// TIA Portal project "PID_PROCCESS_CONTROL" (V16)

(* hardware
DEVICE "S7-1200 station_1"  S7-1200 Station
   slot 0: "Rack_0"  S7-1200 Rack  Rack  V1.0
   slot 1: "PLC_1"  CPU 1214C DC/DC/DC  6ES7 214-1AG40-0XB0  V4.4
   slot 2: "AI 4x13BIT/AQ 2x14BIT_1"  6ES7 234-4HE32-0XB0  V2.1
*)

// ===== PLC "PLC_1"  CPU 1214C DC/DC/DC =====

VAR_GLOBAL   // PLC tag table "Default tag table"
   "Tag_1" AT %MD2 : DWord;
   "Tag_2" AT %M500.0 : Bool;
   "Tag_3" AT %MD67 : Real;
   "Tag_4" AT %MD77 : DWord;
   "SP" AT %MD96 : Real;
   "Tag_5" AT %Q0.3 : Bool;
   "Tag_6" AT %MD70 : Real;
END_VAR

VAR_GLOBAL   // PLC tag table "INPUTS&OUTPUTS"
   "PRESSURE_SENSOR" AT %IW64 : Int;
   "FLOW_VALVE" AT %QW96 : Int;
   "SWITCH_1" AT %I0.1 : Bool;
   "SWITCH_2_SOLENOID" AT %I0.2 : Bool;
   "PUMP" AT %Q0.0 : Bool;
   "SOLENOID" AT %Q0.1 : Bool;
   "STORE_MEM" AT %MD20 : DWord;
   "FINAL_VAL" AT %MD30 : DWord;
END_VAR

ORGANIZATION_BLOCK "Main"   // OB1, LAD, ProgramCycle
TITLE = "Main Program Sweep (Cycle)"
{ S7_Optimized_Access := 'TRUE' }
VERSION : 0.1
   VAR_INPUT
      Initial_Call : Bool;   // Initial call of this OB
      Remanence : Bool;   // =True, if remanent data are available
   END_VAR
BEGIN

REGION Network 1
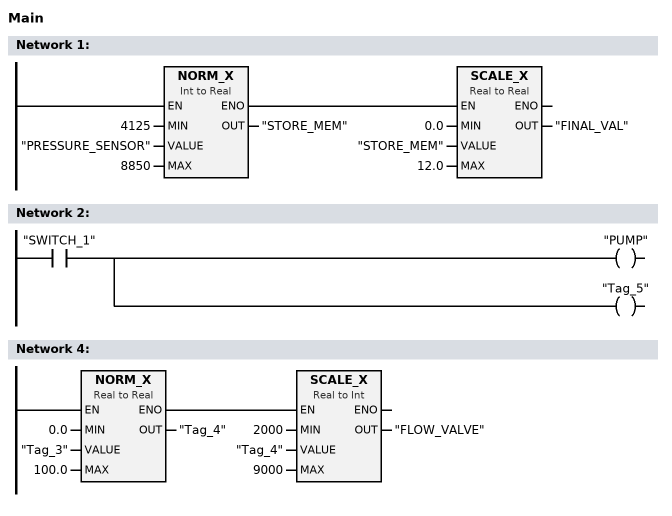
   RUNG wire#powerrail
      { S7_Templates := "[SrcType := Int, DestType := Real]" } Normalize(min := 4125, value := "PRESSURE_SENSOR", max := 8850, out => "STORE_MEM")
      { S7_Templates := "[SrcType := Real, DestType := Real]" } Scale(min := 0.0, value := "STORE_MEM", max := 12.0, out => "FINAL_VAL")
   END_RUNG
   // the same network as SCL:
   "STORE_MEM" := NORM_X(MIN := 4125, VALUE := "PRESSURE_SENSOR", MAX := 8850);
   "FINAL_VAL" := SCALE_X(MIN := 0.0, VALUE := "STORE_MEM", MAX := 12.0);
END_REGION

REGION Network 2
   RUNG wire#powerrail
      Contact( "SWITCH_1" )
      wire#w1
      Coil( "PUMP" )
   END_RUNG
   RUNG wire#w1
      Coil( "Tag_5" )
   END_RUNG
   // the same network as SCL:
   "PUMP" := "SWITCH_1";
   "Tag_5" := "SWITCH_1";
END_REGION

REGION Network 4
   RUNG wire#powerrail
      { S7_Templates := "[SrcType := Real, DestType := Real]" } Normalize(min := 0.0, value := "Tag_3", max := 100.0, out => "Tag_4")
      { S7_Templates := "[SrcType := Real, DestType := Int]" } Scale(min := 2000, value := "Tag_4", max := 9000, out => "FLOW_VALVE")
   END_RUNG
   // the same network as SCL:
   "Tag_4" := NORM_X(MIN := 0.0, VALUE := "Tag_3", MAX := 100.0);
   "FLOW_VALVE" := SCALE_X(MIN := 2000, VALUE := "Tag_4", MAX := 9000);
END_REGION
END_ORGANIZATION_BLOCK

ORGANIZATION_BLOCK "Cyclic interrupt"   // OB30, LAD, CyclicInterrupt
{ S7_Optimized_Access := 'TRUE' }
VERSION : 0.1
   VAR_INPUT
      Initial_Call : Bool;   // Initial call of this OB
      Event_Count : Int;   // Events discarded
   END_VAR
BEGIN
END_ORGANIZATION_BLOCK

ORGANIZATION_BLOCK "TRIAL"   // OB31, LAD, CyclicInterrupt
{ S7_Optimized_Access := 'TRUE' }
VERSION : 0.1
   VAR_INPUT
      Initial_Call : Bool;   // Initial call of this OB
      Event_Count : Int;   // Events discarded
   END_VAR
BEGIN

REGION Network 1
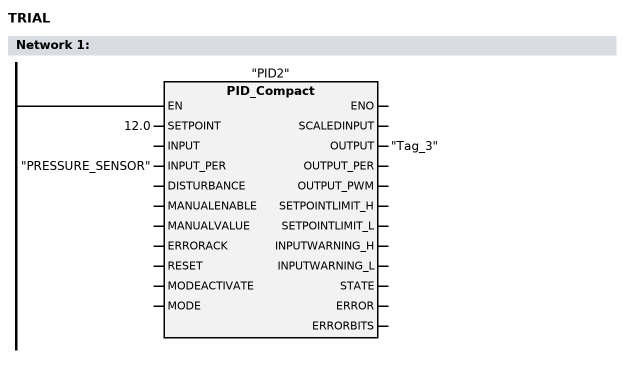
   "PID2"(Setpoint := 12.0, Input_PER := "PRESSURE_SENSOR", Output => "Tag_3");   // PID_Compact
END_REGION
END_ORGANIZATION_BLOCK